FUNCTION_BLOCK PUBLIC FB_DevValve EXTENDS FB_DevBase
VAR_INPUT
	// Manual control 
	stManualCtrl	: UDT_ManualValveControl ;
END_VAR
VAR_OUTPUT
	// ===== Status indicators =======
	bFco_Closed		:	BOOL := FALSE ;
	bFco_Open		: 	BOOL := FALSE ;
END_VAR
VAR
	// Pararmeters
		stParTimeToClose	: Udt_Parameter := (fValue := 50) ; // time to close parameter
		stParTimeToOpen		: Udt_Parameter	:= (fValue := 50) ; // Time to open parameter
	// Hardware links 
		q_Open			AT %Q* : BOOL := FALSE 	; // Open valve
		q_Close 		AT %Q* : BOOL := FALSE	; // Close valve
	// Internal commands
		bCmdClose 	: BOOL := FALSE ; // close valve 
		bCmdOpen	: BOOL := FALSE ; // Open valve
		bCmdHold	: BOOL := FALSE ; // Hold valve status change
	// Time functions 
		fbTOnClose	: TON	; // Timer for valve close
		FbTOnOpen	: TON 	; // Timer for valve Open
		fbTimerSwitchDir: TON ; // Time for teach function switch direction 
	// reset and safe state
		eResetState		: E_ValveResetState := 0		; // Cylinder reset state variable (default is idle) 
		eSafeState		: E_ValveResetState	:= 0		; // Valve safe state
END_VAR

// set device type
IF eDevType = E_Devices.Undefined THEN 
	eDevType := E_Devices.Valve ;
END_IF

// Call base function
SUPER^();

// ===== hold all actions if not initialized ======
IF NOT bInitOk THEN
	RETURN;
END_IF 

// ====== Set Outputs =======
	ExecSetOutPuts();

// ===== collect feedback ======
	ExecSetFeedback();

METHOD PUBLIC CmdClose : BOOL // close valve or retract cylinder
VAR_INPUT
END_VAR
// ====== Set close command if enabled ======
	bCmdClose 	:= TRUE	;		
	bCmdOpen 	:= FALSE;
	
// ===== Set feedback ======
	CmdClose := bFco_Closed ;
END_METHOD

METHOD PUBLIC CmdHold : BOOL
VAR_INPUT
END_VAR
// ====== set hold command =====
	bCmdHold := TRUE ;

CmdHold := bBlockedCommand ;
END_METHOD

METHOD PUBLIC CmdManual : BOOL
VAR_IN_OUT
END_VAR
// Enable manual commands
bCmdManual S= TRUE ;

// execute manual command 
	IF stManualCtrl.bCmdOpen THEN 
		CmdOpen();
	ELSIF stManualCtrl.bCmdClose THEN 
	 	CmdClose(); 
	ELSIF stManualCtrl.bCmdTeach THEN
		CmdTeach ();
	END_IF
END_METHOD

METHOD PUBLIC CmdOpen : BOOL // Open valve or retract cylinder
VAR_INPUT
END_VAR
// ====== Set open command if enabled ======
	bCmdClose 	:= FALSE;		
	bCmdOpen 	:= TRUE	;
	
// ===== Set feedback ======
	CmdOpen := bFco_Open ;
END_METHOD

METHOD CmdReset : BOOL
VAR_INPUT
END_VAR
// ====== Set outputs according to reset state =======
	IF bEnable THEN 
		CASE eResetState OF 
			E_ValveResetState.Res_Idle:
				bCmdClose 	:= FALSE;		
				bCmdOpen 	:= FALSE;
			E_ValveResetState.Res_Closed:
				bCmdClose 	:= TRUE	;		
				bCmdOpen 	:= FALSE;
			E_ValveResetState.Res_Open:
				bCmdClose 	:= FALSE;		
				bCmdOpen 	:= TRUE	;
		ELSE
			;
		END_CASE
	END_IF
// ======= Reset Error bit ======
	bErrorActive 	:= FALSE;
	bBussy			:= FALSE;
END_METHOD

METHOD PUBLIC CmdSafeStop : BOOL
VAR_INPUT
END_VAR
CASE eSafeState OF 
	E_ValveResetState.Res_Idle:
		bDevIsSafe := bFco_Closed OR bFco_Open ;
	E_ValveResetState.Res_Closed:
		bDevIsSafe := bFco_Closed ;
	E_ValveResetState.Res_Open:
		bDevIsSafe := bFco_Open ;
END_CASE

CmdSafeStop := bDevIsSafe OR NOT bInitOk ;
END_METHOD

METHOD PUBLIC CmdTeach : BOOL
VAR_INPUT
END_VAR
// ====== teach cylinder from hardware inputs ======
	fbTimerSwitchDir(PT:= T#1S); 
// ===== Start test loop =====
IF bFco_Closed AND fbTimerSwitchDir.Q THEN
	bCmdClose 			:= FALSE;
	bCmdOpen 			:= TRUE ;
	fbTimerSwitchDir.IN	:= FALSE; 
ELSIF bFco_Open AND fbTimerSwitchDir.Q THEN
	bCmdClose 			:= TRUE ;
	bCmdOpen 			:= FALSE;
	fbTimerSwitchDir.IN	:= FALSE; 
ELSIF NOT bCmdClose AND NOT bCmdOpen THEN 
	bCmdClose 			:= TRUE ;
	bCmdOpen 			:= FALSE;
END_IF

// ====== start timing ========
	IF bCmdClose AND bFco_Closed THEN 
		fbTimerSwitchDir.IN := TRUE 		;
	ELSIF bCmdOpen AND bFco_Open THEN 
		fbTimerSwitchDir.IN := TRUE 		;
	END_IF
END_METHOD

METHOD PROTECTED ExecSetFeedback : BOOL
VAR_INPUT
END_VAR
// ====== Set timers =======
	fbTOnClose	(PT 	:= LREAL_TO_TIME(stParTimeToClose.fValue))	;
	FbTOnOpen	(PT		:= LREAL_TO_TIME(stParTimeToOpen.fValue))	;

// ====== Set timed feedback ======
	IF q_Close THEN 
		fbTOnClose.IN 	:= TRUE ;
		fbTOnopen.IN 	:= FALSE;
	ELSIF q_Open THEN 
		fbTOnClose.IN 	:= FALSE;
		FbTOnOpen.IN	:= TRUE ;
	ELSE 
		fbTOnClose.IN 	:= FALSE;
		FbTOnOpen.IN	:= FALSE;
	END_IF
	
// ====== set outputs =======
	bFco_Closed := fbTOnClose.Q ;
	bFco_Open	:= FbTOnOpen.Q	;
	bReady		:= bFco_Closed OR bFco_Open ;
END_METHOD

METHOD PROTECTED ExecSetOutPuts : BOOL
VAR_INPUT
END_VAR
// ======= Set Outputs according to commands and check safety features =======
IF bSafetyOk THEN
	IF NOT bCmdHold AND (bEnable OR bCmdManual) THEN  
		q_Close	:= bCmdClose;
		q_Open	:= bCmdOpen	;
		bBlockedCommand := FALSE ;
	ELSE
		bBlockedCommand := TRUE ;
	END_IF
ELSE
	CASE eSafeState OF 
		E_ValveResetState.Res_Idle:
			q_Close	:= bFco_Closed;		
			q_Open 	:= bFco_Open;
		E_ValveResetState.Res_Closed:
			q_Close	:= TRUE	;		
			q_Open 	:= FALSE;
		E_ValveResetState.Res_Open:
			q_Close	:= FALSE;		
			q_Open 	:= TRUE	;
	END_CASE
	bCmdClose 	:= bFco_Closed 	;
	bCmdOpen	:= bFco_Open	;
	
END_IF

// Reset manual and hold commands
bCmdHold 	:= FALSE ;
bCmdManual 	:= FALSE ;
END_METHOD

METHOD PUBLIC Init : BOOL
VAR_INPUT
	// Valve data 
	nDevNumber	: UDINT				:= 0		; // Cylinder identification number
	// Command state
	eResetState		: E_ValveResetState := 0		; // Cylinder reset state variable (default is idle) 
	eSafeState		: E_ValveResetState	:= 0		; // Valve safe state
END_VAR
// ====== Calculate device id =====
	THIS^.nDevNumber := nDevNumber ;
	SUPER^.CalcDeviceId();
// ====== Set message information =======
	stFault.ComponentType	:= E_ComponentTypes.Cylinder 		;
	
// ====== Set outputs according to reset state =======
	THIS^.eResetState 	:= eResetState 	;
	THIS^.eSafeState	:= eSafeState	;	

	IF bEnable THEN 
		CASE eResetState OF 
			E_ValveResetState.Res_Idle:
				bCmdClose 	:= bFco_Closed	;		
				bCmdOpen 	:= bFco_Open	;
			E_ValveResetState.Res_Closed:
				bCmdClose 	:= TRUE;		
				bCmdOpen 	:= FALSE;
			E_ValveResetState.Res_Open:
				bCmdClose 	:= FALSE;		
				bCmdOpen 	:= TRUE ;
		END_CASE
	END_IF
// ======= Reset Error bit ======
	bErrorActive 	:= FALSE;
	bBussy			:= FALSE;

// ===== Set device type for manual control =====
	eDevType := E_Devices.Valve ;
	
// ===== configure parameters =====
	stParTimeToClose.fMinimum 		:= 0 		;
	stParTimeToClose.fMaximum		:= 60000 	;
	stParTimeToClose.nNumber 		:= nDevId + 1;
	stParTimeToClose.sDiscription  	:= CONCAT( STR1 := sDevName, STR2 := 'avarage time it takes for the valve to close in miliseconds');
	stParTimeToClose.sName			:= CONCAT( STR1 := sDevName, STR2 := 'time to close');
	stParTimeToClose.sType			:= 'CPar';
	stParTimeToClose.sUnit			:= 'ms';

	stParTimeToOpen.fMinimum 		:= 0 		;
	stParTimeToOpen.fMaximum		:= 60000 	;
	stParTimeToOpen.nNumber 		:= nDevId + 2;
	stParTimeToOpen.sDiscription  	:= CONCAT( STR1 := sDevName, STR2 := 'avarage time it takes for the valve to open in miliseconds');
	stParTimeToOpen.sName			:= CONCAT( STR1 := sDevName, STR2 := 'time to open');
	stParTimeToOpen.sType			:= 'CPar';
	stParTimeToOpen.sUnit			:= 'ms';
	
	// add parameters to handler 
	refFbParHandler.CmdAddParameter( refParameter := stParTimeToClose );
	refFbParHandler.CmdAddParameter( refParameter := stParTimeToOpen );
	
// ====== Set init status bit =======
	bInitOk := TRUE ;
END_METHOD

END_FUNCTION_BLOCK

(* stored: Version 1.1.0.1, ProductVersion 3.1.4024.5
   POU FB_DevValve: Id {ba396402-0ac8-4d5d-a8f4-911b90a2c3dc}, SpecialFunc None
   Folder Private: Id {2dd80cd9-fe6b-4d89-aae3-48132b1585a9}
   Method CmdClose: Id {a782a9c4-fe6c-4821-bc15-4a5b2458d528}
   Method CmdHold: Id {af07192d-9229-4e2b-8dd0-febfb84d4f3e}
   Method CmdManual: Id {e0148156-b539-4a27-871c-4550f6ffb60a}
   Method CmdOpen: Id {54b61d17-85d8-43fc-a979-9c7d65147693}
   Method CmdReset: Id {f243310c-6787-45be-b839-74681681062f}
   Method CmdSafeStop: Id {e95074f6-7b45-0ac3-1b01-bd35092d95b2}
   Method CmdTeach: Id {3f2593c7-29ea-0862-082c-1fa6f192418d}
   Method ExecSetFeedback: Id {bec6c7c2-5e23-47f9-8f90-22cbd47ce8f5}
   Method ExecSetOutPuts: Id {c7a194a0-0cdb-4788-8c09-c5fb927df87c}
   Method Init: Id {b8e244d6-5d8d-4fc7-8d11-89f2fc179f0b} *)
